// TIA Portal project "TRAFFIC_LIGHTS_BRIDGE_CROSSING_SCL_BASIC" (V19)

(* hardware
DEVICE "S7-1200 station_1"  S7-1200 Station
   slot 0: "Rack_0"  S7-1200 Rack  Rack  V1.0
   slot 1: "TRAFFIC_LIGHTS_PLC"  CPU 1215C DC/DC/DC  6ES7 215-1AG40-0XB0  V4.6
*)

// ===== PLC "TRAFFIC_LIGHTS_PLC"  CPU 1215C DC/DC/DC =====

VAR_GLOBAL   // PLC tag table "System_Tags"
   "Clock_Byte" AT %MB0 : Byte;
   "Clock_10Hz" AT %M0.0 : Bool;
   "Clock_5Hz" AT %M0.1 : Bool;
   "Clock_2.5Hz" AT %M0.2 : Bool;
   "Clock_2Hz" AT %M0.3 : Bool;
   "Clock_1.25Hz" AT %M0.4 : Bool;
   "Clock_1Hz" AT %M0.5 : Bool;
   "Clock_0.625Hz" AT %M0.6 : Bool;
   "Clock_0.5Hz" AT %M0.7 : Bool;
   "System_Byte" AT %MB1 : Byte;
   "FirstScan" AT %M1.0 : Bool;
   "DiagStatusUpdate" AT %M1.1 : Bool;
   "AlwaysTRUE" AT %M1.2 : Bool;
   "AlwaysFALSE" AT %M1.3 : Bool;
END_VAR

VAR_GLOBAL   // PLC tag table "PLC_Inputs"
   "DI0.0" AT %I0.0 : Bool;   // Digital Input
   "DI0.1" AT %I0.1 : Bool;   // Digital Input
   "DI0.2" AT %I0.2 : Bool;   // Digital Input
   "DI0.3" AT %I0.3 : Bool;   // Digital Input
   "DI0.4" AT %I0.4 : Bool;   // Digital Input
   "DI0.5" AT %I0.5 : Bool;   // Digital Input
   "DI0.6" AT %I0.6 : Bool;   // Digital Input
   "DI0.7" AT %I0.7 : Bool;   // Digital Input
   "DI1.0" AT %I1.0 : Bool;   // Digital Input
   "DI1.1" AT %I1.1 : Bool;   // Digital Input
   "DI1.2" AT %I1.2 : Bool;   // Digital Input
   "DI1.3" AT %I1.3 : Bool;   // Digital Input
   "DI1.4" AT %I1.4 : Bool;   // Digital Input
   "DI1.5" AT %I1.5 : Bool;   // Digital Input
   "AI0.0" AT %IW64 : Word;   // Analog Input
   "AI0.1" AT %IW66 : Word;   // Analog Input
END_VAR

VAR_GLOBAL   // PLC tag table "PLC_Outputs"
   "DQ0.0" AT %Q0.0 : Bool;   // Digital Output
   "DQ0.1" AT %Q0.1 : Bool;   // Digital Output
   "DQ0.2" AT %Q0.2 : Bool;   // Digital Output
   "DQ0.3" AT %Q0.3 : Bool;   // Digital Output
   "DQ0.4" AT %Q0.4 : Bool;   // Digital Output
   "DQ0.5" AT %Q0.5 : Bool;   // Digital Output
   "DQ0.6" AT %Q0.6 : Bool;   // Digital Output
   "DQ0.7" AT %Q0.7 : Bool;   // Digital Output
   "DQ1.0" AT %Q1.0 : Bool;   // Digital Output
   "DQ1.1" AT %Q1.1 : Bool;   // Digital Output
   "AQ0.0" AT %QW64 : Word;   // Analog Output
   "AQ0.1" AT %QW66 : Word;   // Analog Output
END_VAR

VAR_GLOBAL   // PLC tag table "Trigger_Tags"
   "xAmberTOF_Trig" AT %M2.0 : Bool;
   "xTrig2" AT %M2.1 : Bool;
   "xTrig3" AT %M2.2 : Bool;
   "xTrig4" AT %M2.3 : Bool;
   "xTrig5" AT %M2.4 : Bool;
END_VAR

// folder: WS01_TVET_Workstation/00-I/O_Mapping

DATA_BLOCK "DB001-PLC_I/O"   // DB1
{ S7_Optimized_Access := 'TRUE' }
VERSION : 0.1
   VAR
      PLC_Inputs : Struct   // PLC Inputs Structure
         "xDI0.0" : Bool;
         "xDI0.1" : Bool;
         "xDI0.2" : Bool;
         "xDI0.3" : Bool;
         "xDI0.4" : Bool;
         "xDI0.5" : Bool;
         "xDI0.6" : Bool;
         "xDI0.7" : Bool;
         "xDI1.0" : Bool;
         "xDI1.1" : Bool;
         "xDI1.2" : Bool;
         "xDI1.3" : Bool;
         "xDI1.4" : Bool;
         "xDI1.5" : Bool;
         "iAI0.0_Scalled" : Int;
         "iAI0.1_Scalled" : Int;
      END_STRUCT;
      PLC_Outputs : Struct   // PLC Outputs Structure
         xLeft_GreenLED : Bool;   // Left Side Green LED
         xLeft_AmberLED : Bool;   // Left Side Amber LED
         xLeft_RedLED : Bool;   // Left Side Red LED
         xRight_GreenLED : Bool;   // Right Side Green LED
         xRight_AmberLED : Bool;   // Right Side Amber LED
         xRight_RedLED : Bool;   // Right Side Red LED
         "xDQ0.6" : Bool;
         "xDQ0.7" : Bool;
         "xDQ1.0" : Bool;
         "xDQ1.1" : Bool;
         "iAQ0.0" : Int;
         "iAQ0.1" : Int;
      END_STRUCT;
   END_VAR
BEGIN
END_DATA_BLOCK

// folder: WS01_TVET_Workstation/01-Traffic_Logic

DATA_BLOCK "FB001-Traffic_Control_DB"   // DB2
{ S7_Optimized_Access := 'TRUE' }
VERSION : 0.1
// stored: InstanceOfName FB001-Traffic_Control
"FB001-Traffic_Control"
BEGIN
END_DATA_BLOCK

// folder: (top level)

ORGANIZATION_BLOCK "Main"   // OB1, LAD, ProgramCycle
TITLE = "Main Program Sweep (Cycle)"
{ S7_Optimized_Access := 'TRUE' }
VERSION : 0.1
   VAR_INPUT
      Initial_Call : Bool;   // Initial call of this OB
      Remanence : Bool;   // =True, if remanent data are available
   END_VAR
BEGIN

REGION Network 1 (SCL): ================= PROGRAM_INFORMATION =================
   (*
   =================================================================
   ***** TRAFFIC LIGHTS - BRIDGE CROSSING WITHOUT PUSH BUTTONS *****
   =================================================================

   TVET Workstation WS01
   - 1215C DC/DC/DC - 6ES7215-1AG40-0XB0
   - IP:       192.168.0.175/24
   - Gateway:  192.168.0.1

   =======================================================================

   The program has 2 main sections - I/O Handler & Traffic Control.

   I/O Handler FC:
   We are directly interacting with the PLC's I/O and DB tags, therefore
   a FC can be used for the I/O mapping logic.
   - maps the physical inputs & outputs to corresponding tags in DB001
     (this makes code easier to read, maintain & troubleshoot).

   Traffic Control FB:
   We use a FB for traffic control logic as any additional tags needed can
   be created in the FB interface.
   - sets the default state of the system at startup,
   - make use of SCL state machine & timers to automatically change LED
     states in a loop.

   Additional Notes:
   PLC Tags have been grouped relating to their use/function.

   =======================================================================
   *)
END_REGION

REGION Network 2: ================= I/O_HANDLING =================
   // > Call the PLC I/O Handler Function
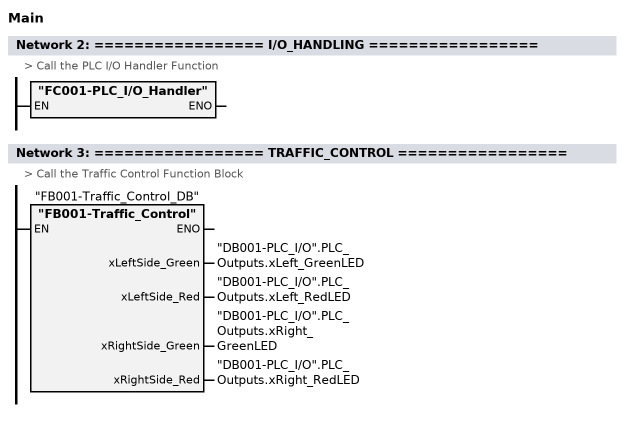
   RUNG wire#powerrail
      "FC001-PLC_I/O_Handler"()
   END_RUNG
   // the same network as SCL:
   "FC001-PLC_I/O_Handler"();
END_REGION

REGION Network 3: ================= TRAFFIC_CONTROL =================
   // > Call the Traffic Control Function Block
   RUNG wire#powerrail
      "FB001-Traffic_Control_DB"(xLeftSide_Green => "DB001-PLC_I/O".PLC_Outputs.xLeft_GreenLED, xLeftSide_Red => "DB001-PLC_I/O".PLC_Outputs.xLeft_RedLED, xRightSide_Green => "DB001-PLC_I/O".PLC_Outputs.xRight_GreenLED, xRightSide_Red => "DB001-PLC_I/O".PLC_Outputs.xRight_RedLED)
   END_RUNG
   // the same network as SCL:
   "FB001-Traffic_Control_DB"(xLeftSide_Green => "DB001-PLC_I/O".PLC_Outputs.xLeft_GreenLED,   // "FB001-Traffic_Control"
                           xLeftSide_Red => "DB001-PLC_I/O".PLC_Outputs.xLeft_RedLED,
                           xRightSide_Green => "DB001-PLC_I/O".PLC_Outputs.xRight_GreenLED,
                           xRightSide_Red => "DB001-PLC_I/O".PLC_Outputs.xRight_RedLED);
END_REGION
END_ORGANIZATION_BLOCK

// folder: WS01_TVET_Workstation/00-I/O_Mapping

FUNCTION "FC001-PLC_I/O_Handler" : Void   // FC1, LAD
{ S7_Optimized_Access := 'TRUE' }
VERSION : 0.1
   VAR_TEMP
      "rAI0.0_Temp" : Real;   // -
      "rAI0.1_Temp" : Real;   // -
      "rAQ0.0_Temp" : Real;   // -
      "rAQ0.1_Temp" : Real;   // -
   END_VAR
BEGIN

REGION Network 1: ================= DIGITAL_INPUTS =================
END_REGION

REGION Network 2: BANK_0
   // > DI0.0 - DI0.7
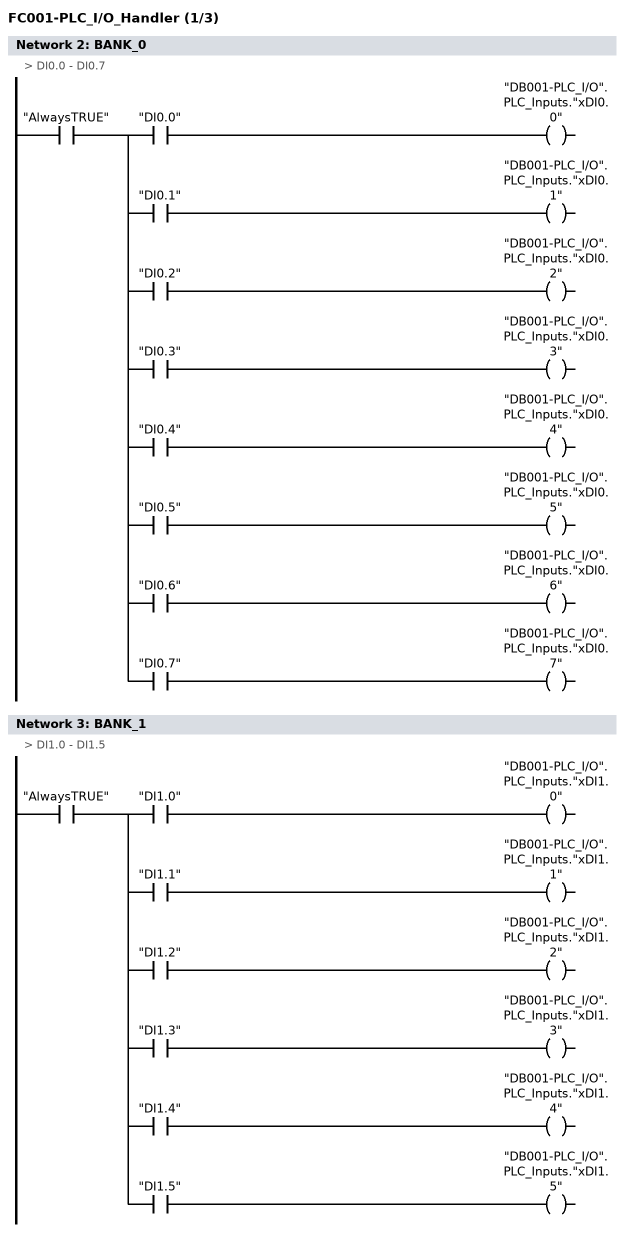
   RUNG wire#powerrail
      Contact( "AlwaysTRUE" )
      wire#w1
      Contact( "DI0.0" )
      Coil( "DB001-PLC_I/O".PLC_Inputs."xDI0.0" )
   END_RUNG
   RUNG wire#w1
      Contact( "DI0.1" )
      Coil( "DB001-PLC_I/O".PLC_Inputs."xDI0.1" )
   END_RUNG
   RUNG wire#w1
      Contact( "DI0.2" )
      Coil( "DB001-PLC_I/O".PLC_Inputs."xDI0.2" )
   END_RUNG
   RUNG wire#w1
      Contact( "DI0.3" )
      Coil( "DB001-PLC_I/O".PLC_Inputs."xDI0.3" )
   END_RUNG
   RUNG wire#w1
      Contact( "DI0.4" )
      Coil( "DB001-PLC_I/O".PLC_Inputs."xDI0.4" )
   END_RUNG
   RUNG wire#w1
      Contact( "DI0.5" )
      Coil( "DB001-PLC_I/O".PLC_Inputs."xDI0.5" )
   END_RUNG
   RUNG wire#w1
      Contact( "DI0.6" )
      Coil( "DB001-PLC_I/O".PLC_Inputs."xDI0.6" )
   END_RUNG
   RUNG wire#w1
      Contact( "DI0.7" )
      Coil( "DB001-PLC_I/O".PLC_Inputs."xDI0.7" )
   END_RUNG
   // the same network as SCL:
   "DB001-PLC_I/O".PLC_Inputs."xDI0.0" := "AlwaysTRUE" AND "DI0.0";
   "DB001-PLC_I/O".PLC_Inputs."xDI0.1" := "AlwaysTRUE" AND "DI0.1";
   "DB001-PLC_I/O".PLC_Inputs."xDI0.2" := "AlwaysTRUE" AND "DI0.2";
   "DB001-PLC_I/O".PLC_Inputs."xDI0.3" := "AlwaysTRUE" AND "DI0.3";
   "DB001-PLC_I/O".PLC_Inputs."xDI0.4" := "AlwaysTRUE" AND "DI0.4";
   "DB001-PLC_I/O".PLC_Inputs."xDI0.5" := "AlwaysTRUE" AND "DI0.5";
   "DB001-PLC_I/O".PLC_Inputs."xDI0.6" := "AlwaysTRUE" AND "DI0.6";
   "DB001-PLC_I/O".PLC_Inputs."xDI0.7" := "AlwaysTRUE" AND "DI0.7";
END_REGION

REGION Network 3: BANK_1
   // > DI1.0 - DI1.5
   RUNG wire#powerrail
      Contact( "AlwaysTRUE" )
      wire#w1
      Contact( "DI1.0" )
      Coil( "DB001-PLC_I/O".PLC_Inputs."xDI1.0" )
   END_RUNG
   RUNG wire#w1
      Contact( "DI1.1" )
      Coil( "DB001-PLC_I/O".PLC_Inputs."xDI1.1" )
   END_RUNG
   RUNG wire#w1
      Contact( "DI1.2" )
      Coil( "DB001-PLC_I/O".PLC_Inputs."xDI1.2" )
   END_RUNG
   RUNG wire#w1
      Contact( "DI1.3" )
      Coil( "DB001-PLC_I/O".PLC_Inputs."xDI1.3" )
   END_RUNG
   RUNG wire#w1
      Contact( "DI1.4" )
      Coil( "DB001-PLC_I/O".PLC_Inputs."xDI1.4" )
   END_RUNG
   RUNG wire#w1
      Contact( "DI1.5" )
      Coil( "DB001-PLC_I/O".PLC_Inputs."xDI1.5" )
   END_RUNG
   // the same network as SCL:
   "DB001-PLC_I/O".PLC_Inputs."xDI1.0" := "AlwaysTRUE" AND "DI1.0";
   "DB001-PLC_I/O".PLC_Inputs."xDI1.1" := "AlwaysTRUE" AND "DI1.1";
   "DB001-PLC_I/O".PLC_Inputs."xDI1.2" := "AlwaysTRUE" AND "DI1.2";
   "DB001-PLC_I/O".PLC_Inputs."xDI1.3" := "AlwaysTRUE" AND "DI1.3";
   "DB001-PLC_I/O".PLC_Inputs."xDI1.4" := "AlwaysTRUE" AND "DI1.4";
   "DB001-PLC_I/O".PLC_Inputs."xDI1.5" := "AlwaysTRUE" AND "DI1.5";
END_REGION

REGION Network 4: ================= DIGITAL_OUTPUTS =================
END_REGION

REGION Network 5: BANK_0
   // > DQ0.0 - DQ0.7
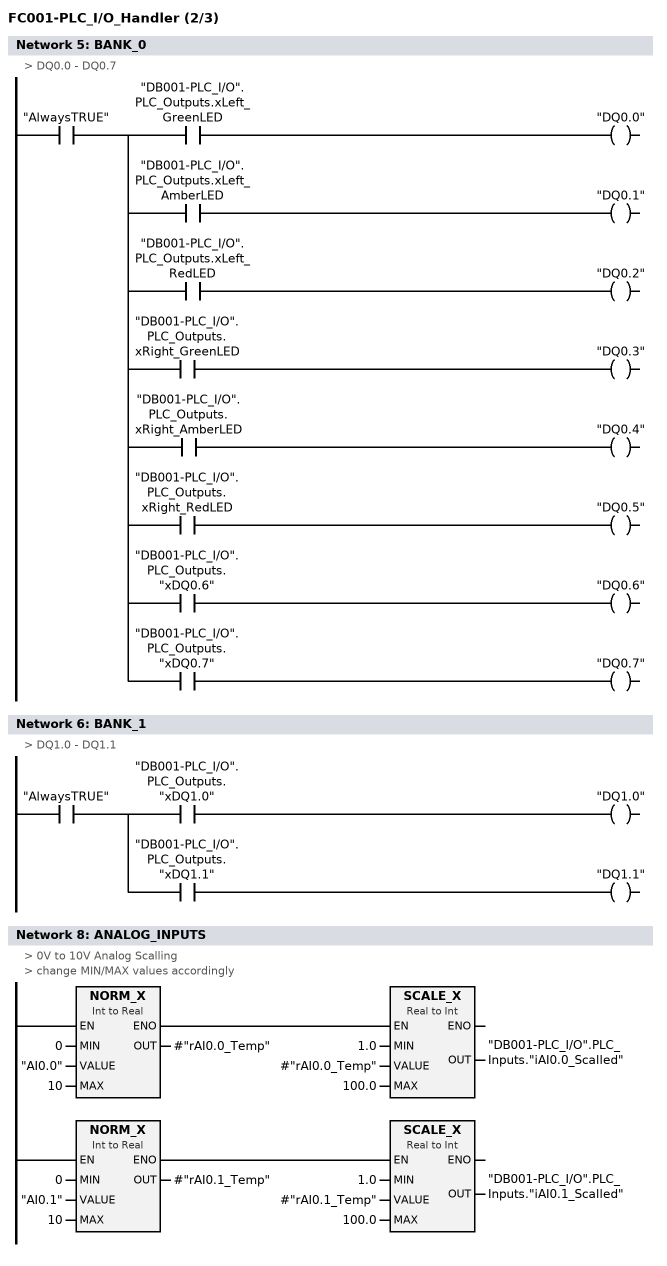
   RUNG wire#powerrail
      Contact( "AlwaysTRUE" )
      wire#w1
      Contact( "DB001-PLC_I/O".PLC_Outputs.xLeft_GreenLED )
      Coil( "DQ0.0" )
   END_RUNG
   RUNG wire#w1
      Contact( "DB001-PLC_I/O".PLC_Outputs.xLeft_AmberLED )
      Coil( "DQ0.1" )
   END_RUNG
   RUNG wire#w1
      Contact( "DB001-PLC_I/O".PLC_Outputs.xLeft_RedLED )
      Coil( "DQ0.2" )
   END_RUNG
   RUNG wire#w1
      Contact( "DB001-PLC_I/O".PLC_Outputs.xRight_GreenLED )
      Coil( "DQ0.3" )
   END_RUNG
   RUNG wire#w1
      Contact( "DB001-PLC_I/O".PLC_Outputs.xRight_AmberLED )
      Coil( "DQ0.4" )
   END_RUNG
   RUNG wire#w1
      Contact( "DB001-PLC_I/O".PLC_Outputs.xRight_RedLED )
      Coil( "DQ0.5" )
   END_RUNG
   RUNG wire#w1
      Contact( "DB001-PLC_I/O".PLC_Outputs."xDQ0.6" )
      Coil( "DQ0.6" )
   END_RUNG
   RUNG wire#w1
      Contact( "DB001-PLC_I/O".PLC_Outputs."xDQ0.7" )
      Coil( "DQ0.7" )
   END_RUNG
   // the same network as SCL:
   "DQ0.0" := "AlwaysTRUE" AND "DB001-PLC_I/O".PLC_Outputs.xLeft_GreenLED;
   "DQ0.1" := "AlwaysTRUE" AND "DB001-PLC_I/O".PLC_Outputs.xLeft_AmberLED;
   "DQ0.2" := "AlwaysTRUE" AND "DB001-PLC_I/O".PLC_Outputs.xLeft_RedLED;
   "DQ0.3" := "AlwaysTRUE" AND "DB001-PLC_I/O".PLC_Outputs.xRight_GreenLED;
   "DQ0.4" := "AlwaysTRUE" AND "DB001-PLC_I/O".PLC_Outputs.xRight_AmberLED;
   "DQ0.5" := "AlwaysTRUE" AND "DB001-PLC_I/O".PLC_Outputs.xRight_RedLED;
   "DQ0.6" := "AlwaysTRUE" AND "DB001-PLC_I/O".PLC_Outputs."xDQ0.6";
   "DQ0.7" := "AlwaysTRUE" AND "DB001-PLC_I/O".PLC_Outputs."xDQ0.7";
END_REGION

REGION Network 6: BANK_1
   // > DQ1.0 - DQ1.1
   RUNG wire#powerrail
      Contact( "AlwaysTRUE" )
      wire#w1
      Contact( "DB001-PLC_I/O".PLC_Outputs."xDQ1.0" )
      Coil( "DQ1.0" )
   END_RUNG
   RUNG wire#w1
      Contact( "DB001-PLC_I/O".PLC_Outputs."xDQ1.1" )
      Coil( "DQ1.1" )
   END_RUNG
   // the same network as SCL:
   "DQ1.0" := "AlwaysTRUE" AND "DB001-PLC_I/O".PLC_Outputs."xDQ1.0";
   "DQ1.1" := "AlwaysTRUE" AND "DB001-PLC_I/O".PLC_Outputs."xDQ1.1";
END_REGION

REGION Network 7: ================= ANALOG_PROCESSING =================
END_REGION

REGION Network 8: ANALOG_INPUTS
   // > 0V to 10V Analog Scalling
   // > change MIN/MAX values accordingly
   RUNG wire#powerrail
      { S7_Templates := "[SrcType := Int, DestType := Real]" } Normalize(min := 0, value := "AI0.0", max := 10, out => #"rAI0.0_Temp")
      { S7_Templates := "[SrcType := Real, DestType := Int]" } Scale(min := 1.0, value := #"rAI0.0_Temp", max := 100.0, out => "DB001-PLC_I/O".PLC_Inputs."iAI0.0_Scalled")
   END_RUNG
   RUNG wire#powerrail
      { S7_Templates := "[SrcType := Int, DestType := Real]" } Normalize(min := 0, value := "AI0.1", max := 10, out => #"rAI0.1_Temp")
      { S7_Templates := "[SrcType := Real, DestType := Int]" } Scale(min := 1.0, value := #"rAI0.1_Temp", max := 100.0, out => "DB001-PLC_I/O".PLC_Inputs."iAI0.1_Scalled")
   END_RUNG
   // the same network as SCL:
   #"rAI0.0_Temp" := NORM_X(MIN := 0, VALUE := "AI0.0", MAX := 10);
   "DB001-PLC_I/O".PLC_Inputs."iAI0.0_Scalled" := SCALE_X(MIN := 1.0, VALUE := #"rAI0.0_Temp", MAX := 100.0);
   #"rAI0.1_Temp" := NORM_X(MIN := 0, VALUE := "AI0.1", MAX := 10);
   "DB001-PLC_I/O".PLC_Inputs."iAI0.1_Scalled" := SCALE_X(MIN := 1.0, VALUE := #"rAI0.1_Temp", MAX := 100.0);
END_REGION

REGION Network 9: ANALOG_OUTPUTS
   // > 0V to 10V Analog Scalling
   // > change MIN/MAX values accordingly
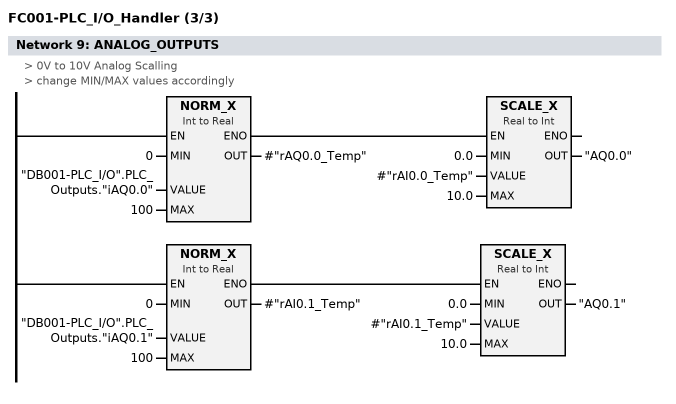
   RUNG wire#powerrail
      { S7_Templates := "[SrcType := Int, DestType := Real]" } Normalize(min := 0, value := "DB001-PLC_I/O".PLC_Outputs."iAQ0.0", max := 100, out => #"rAQ0.0_Temp")
      { S7_Templates := "[SrcType := Real, DestType := Int]" } Scale(min := 0.0, value := #"rAI0.0_Temp", max := 10.0, out => "AQ0.0")
   END_RUNG
   RUNG wire#powerrail
      { S7_Templates := "[SrcType := Int, DestType := Real]" } Normalize(min := 0, value := "DB001-PLC_I/O".PLC_Outputs."iAQ0.1", max := 100, out => #"rAI0.1_Temp")
      { S7_Templates := "[SrcType := Real, DestType := Int]" } Scale(min := 0.0, value := #"rAI0.1_Temp", max := 10.0, out => "AQ0.1")
   END_RUNG
   // the same network as SCL:
   #"rAQ0.0_Temp" := NORM_X(MIN := 0, VALUE := "DB001-PLC_I/O".PLC_Outputs."iAQ0.0", MAX := 100);
   "AQ0.0" := SCALE_X(MIN := 0.0, VALUE := #"rAI0.0_Temp", MAX := 10.0);
   #"rAI0.1_Temp" := NORM_X(MIN := 0, VALUE := "DB001-PLC_I/O".PLC_Outputs."iAQ0.1", MAX := 100);
   "AQ0.1" := SCALE_X(MIN := 0.0, VALUE := #"rAI0.1_Temp", MAX := 10.0);
END_REGION
END_FUNCTION

// folder: WS01_TVET_Workstation/01-Traffic_Logic

FUNCTION_BLOCK "FB001-Traffic_Control"   // FB1, SCL
{ S7_Optimized_Access := 'TRUE' }
VERSION : 0.1
   VAR_OUTPUT
      xLeftSide_Green : Bool;   // Left Side Green LED
      xLeftSide_Red : Bool;   // Left Side Red LED
      xRightSide_Green : Bool;   // Right Side Green LED
      xRightSide_Red : Bool;   // Right Side Red LED
   END_VAR
   VAR
      xFirstScan : Bool;   // First PLC scan catch bit
      iState : Int := 0;   // State number
      TONs : Struct
         tInitial_Delay : TON_TIME;   // Timer ON Delay
         tLeftGreen_Delay : TON_TIME;   // Timer ON Delay
         tLeftRed_Delay : TON_TIME;   // Timer ON Delay
         tRightGreen_Delay : TON_TIME;   // Timer ON Delay
         tRightRed_Delay : TON_TIME;   // Timer ON Delay
      END_STRUCT;
   END_VAR
   VAR CONSTANT
      "3sec" : Time := t#3s;   // PT time constant
      "5sec" : Time := t#5s;   // PT time constant
      "10sec" : Time := t#10s;   // PT time constant
   END_VAR
BEGIN
   REGION OPENING_COMMENTS
       (* 
        * BASIC PROGRAM OPERATION:
        * On startup - both sides start with GREEN LEDs OFF and RED LEDs ON for 5sec.
        *
        * After the initial 5sec has elapsed, left side switches to GREEN ON (RED OFF) for 10sec.
        * After 10sec has elapsed, left side switches to RED ON (GREEN OFF) for 3sec.
        *
        * After 3sec has elapsed, right side switches to GREEN ON (RED OFF) for 10sec.
        * After 10sec has elapsed, right side switches to RED ON (GREEN OFF) for 3sec.
        *
        * Process repeats.
        *
        * STATES:
        * 0 - Both sides RED for 5sec
        * 1 - Left side GREEN & Right side RED for 10sec
        * 2 - Both sides RED for 3 sec (left switch)
        * 3 - Right side GREEN & Left side RED for 10 sec
        * 4 - Both sides RED for 3 sec (right switch)
        *)
   END_REGION


   REGION FIRST_SCAN
       // Catch first PLC scan
       IF "FirstScan" THEN
           #xFirstScan := TRUE;
       END_IF;

       // First PLC scan caught
       IF #xFirstScan THEN
           // Start the inital delay timer & move to the next state
           #TONs.tInitial_Delay(IN := TRUE,     // timer input on
                                PT := #"5sec"); // 5sec duration
           #iState := 0; // initialize the state to 0
       END_IF;
   END_REGION


   REGION STATE_MACHINE
       // LED State Machine
       CASE #iState OF
           0:  // Initial state - both sides red for 5 sec
               #xLeftSide_Green := FALSE;  // left green off
               #xRightSide_Green := FALSE; // right green off
               #xLeftSide_Red := TRUE;     // left red on
               #xRightSide_Red := TRUE;    // right red on

               // Reset xFirstScan flag
               IF #xFirstScan THEN
                   #xFirstScan := FALSE;
               END_IF;

               // Wait for Initial_Delay_TON output
               IF #TONs.tInitial_Delay.Q THEN
                   // Start the left green LED delay timer
                   #TONs.tLeftGreen_Delay(IN := TRUE,      // timer input on
                                          PT := #"10sec"); // 10sec duration
                   // Reset initial timer & move to the next state
                   RESET_TIMER(TIMER := #TONs.tInitial_Delay);
                   #iState := 1;
               END_IF;
               ;
           1:  // Left side green & right side red for 10 sec
               #xLeftSide_Green := TRUE;   // left green on
               #xRightSide_Green := FALSE; // right green off
               #xLeftSide_Red := FALSE;    // left red off
               #xRightSide_Red := TRUE;    // right red on

               // Wait for left green TON ouput
               IF #TONs.tLeftGreen_Delay.Q THEN
                   // Start the left red LED delay timer
                   #TONs.tLeftRed_Delay(IN := TRUE,     // timer input on
                                        PT := #"3sec"); // 3sec duration
                   // Reset left green timer & move to the next state
                   RESET_TIMER(TIMER := #TONs.tLeftGreen_Delay);
                   #iState := 2;
               END_IF;
               ;
           2:  // Both sides red for 3 sec (left switch)
               #xLeftSide_Green := FALSE;  // left green off
               #xRightSide_Green := FALSE; // right green off
               #xLeftSide_Red := TRUE;     // left red on
               #xRightSide_Red := TRUE;    // right red on

               // Wait for left red TON output
               IF #TONs.tLeftRed_Delay.Q THEN
                   // Start the right green LED delay timer
                   #TONs.tRightGreen_Delay(IN := TRUE,      // timer input on
                                           PT := #"10sec"); // 10sec duration
                   // Reset left red timer & move to the next state
                   RESET_TIMER(TIMER := #TONs.tLeftRed_Delay);
                   #iState := 3;
               END_IF;
               ;
           3:  // Right side green & left side red for 10 sec
               #xLeftSide_Green := FALSE; // left green off
               #xRightSide_Green := TRUE; // right green on
               #xLeftSide_Red := TRUE;    // left red on
               #xRightSide_Red := FALSE;  // right red off

               // Wait for right green TON output
               IF #TONs.tRightGreen_Delay.Q THEN
                   // Start the right red LED delay timer
                   #TONs.tRightRed_Delay(IN := TRUE,     // timer input on
                                         PT := #"3sec"); // 3sec duration
                   // Reset right green timer & move to the next state
                   RESET_TIMER(TIMER := #TONs.tRightGreen_Delay);
                   #iState := 4;
               END_IF;
               ;
           4:  // Both sides red for 3 sec (right switch)
               #xLeftSide_Green := FALSE;  // left green off
               #xRightSide_Green := FALSE; // right green off
               #xLeftSide_Red := TRUE;     // left red on
               #xRightSide_Red := TRUE;    // right red on

               // Wait for right red TON output
               IF #TONs.tRightRed_Delay.Q THEN
                   // Start the left green LED delay timer
                   #TONs.tLeftGreen_Delay(IN := TRUE,      // timer input on
                                          PT := #"10sec"); // 10sec duration
                   // Reset right red timer & repeat loop
                   RESET_TIMER(TIMER := #TONs.tRightRed_Delay);
                   #iState := 1; // repeat (move back to state 1)
               END_IF;
               ;
       END_CASE;
   END_REGION
END_FUNCTION_BLOCK